FUNCTION_BLOCK NextVT (* Service Interface Block to switch to the next available VT (Virtual Terminal) *)
  (* Standard: ISO 11783-6; Description: Copyright (c) 2025 Meisterschulen am Ostbahnhof This program and the accompanying materials are made available under the terms of the Eclipse Public License 2.0 which is available at https://www.eclipse.org/legal/epl-2.0/ SPDX-License-Identifier: EPL-2.0 Service Interface Block to switch to the next available VT (Virtual Terminal) This block wraps the functionality of VTC_NextVTButtonPressed() from the ISOBUS driver samples. It allows switching between multiple VTs available on the ISOBUS network. The block performs the following steps: 1. Gets the list of all VTs on the bus using IsoClientsReadListofExtHandles() 2. Finds the currently connected VT using IsoVtcGetStatusInfo(VT_HND) 3. Determines the next VT in the list 4. Switches to the next VT using IsoVtcMultipleNextVT() If there is only one VT on the bus or if the switch fails, an error status is returned. Important: The application must go into a safe state after calling this block as the connection to the current VT will be lost during the transition. *)
  (* Version 1.0, 2025-02-27, Generated, Meisterschulen am Ostbahnhof, initial API and implementation and/or initial documentation *)
  PACKAGE isobus::UT::util;
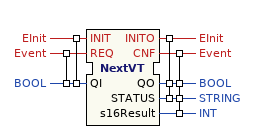
  EVENT_INPUT
    INIT : EInit WITH QI; (* Service Initialization *)
    REQ WITH QI; (* Service Request - Switch to next VT *)
  END_EVENT
  EVENT_OUTPUT
    INITO : EInit WITH QO, STATUS; (* Initialization Confirm *)
    CNF WITH QO, STATUS, s16Result; (* Confirmation - VT switch initiated *)
  END_EVENT
  VAR_INPUT
    QI : BOOL; (* Quality Input - TRUE to enable service *)
  END_VAR
  VAR_OUTPUT
    QO : BOOL; (* Quality Output - TRUE if service executed successfully *)
    STATUS : STRING; (* Service Status *)
    s16Result : INT; (* Return value: 0=E_NO_ERR (success), negative=error code *)
  END_VAR
END_FUNCTION_BLOCK
